// TIA Portal V19 export
VAR_GLOBAL   // PLC tag table "Default tag table"
   A01_Straightener_Ax_Actor_Interface_AddressIn AT %I438.0 : "PD_TEL106_IN";
   A01_Straightener_Ax_Actor_Interface_AddressOut AT %Q438.0 : "PD_TEL106_OUT";
   A02_Carriage_Actor_Interface_AddressIn AT %I408.0 : "PD_TEL106_IN";
   A02_Carriage_Actor_Interface_AddressOut AT %Q408.0 : "PD_TEL106_OUT";
   A02_Rollformer_Actor_Interface_AddressIn AT %I316.0 : "PD_TEL106_IN";
   A02_Rollformer_Actor_Interface_AddressOut AT %Q316.0 : "PD_TEL106_OUT";
   FlyingCarriage_MinStroke AT %I370.0 : Bool;   // 754SQ1 Flying Carriage Minimum Stroke limit switch
   FlyingCarriage_MaxStroke AT %I370.1 : Bool;   // 754SQ1 Flying Carriage Maximum Stroke limit switch
   S120_CU470A1_IN AT %I366.0 : "Tel393In_PM";
   Rollformer_MaxStroke AT %I368.3 : Bool;
   Rollformer_MinStroke AT %I368.2 : Bool;
   Wheel_MeasInput_Interface_Address AT %I369.4 : Bool;
   CutCarriage_MeasuInput_Interface_Address AT %I369.6 : Bool;
   ZeroChk_MeasIn_Interface_Address AT %I369.3 : Bool;
   Weld_MeasInput_Interface_Address AT %I369.0 : Bool;
   Gripper_MeasuInput_Interface_Address AT %I369.5 : Bool;
   CutWheel_MeasInput_Interface_Address AT %I369.7 : Bool;
END_VAR
